PROGRAM MAIN
VAR
END_VAR

METHOD Method1 : BOOL
VAR_INPUT
    nIn1  : INT;
    bIn2  : BOOL;
END_VAR
VAR_OUTPUT
    fOut1 : REAL;
    sOut2 : STRING;
END_VAR
END_METHOD

END_PROGRAM

(* stored: Version 1.1.0.1, ProductVersion 3.1.4024.0
   POU MAIN: Id {d11fd0e5-43eb-4828-b3a1-b1e591b8d394}, SpecialFunc None
   Method Method1: Id {5f08a63b-fa42-4178-a706-0334f7cddc22} *)
